ABB RobotStudio station: Solution1_20200531-184918.rsstn

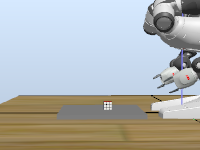
Station Solution1 (saved by RobotStudio 7.0.8746.631)
Controller IRB
  mechanical unit ROB_R: IRB14000_0.5_0.5_R, 6 joints, base frame (0, 0, 0) mm
  mechanical unit ROB_R_7: IRB14000_0.5_0.5_R, 1 joints, base frame (0, 0, 0) mm
  mechanical unit ROB_L: IRB14000_0.5_0.5_L, 6 joints, base frame (0, 0, 0) mm
  mechanical unit ROB_L_7: IRB14000_0.5_0.5_L, 1 joints, base frame (0, 0, 0) mm
Layout (positions relative to the parent item):
  - IRB14000_0.5_0.5 [mechanism, from Robots\IRB14000_0.5_0.5__01.rslib] at (0, 0, 0) mm
  - IRB14000_0.5_0.5_R [mechanism, from Robots\IRB14000_0.5_0.5__01.rslib] at (0, 0, 0) mm; joint values [0, -2.2689, -2.3562, 0.5236, 0, 0.6981, 0] (rad or m)
  - IRB14000_0.5_0.5_L [mechanism, from Robots\IRB14000_0.5_0.5__01.rslib] at (0, 0, 0) mm; joint values [0, -2.2689, 2.3562, 0.5236, 0, 0.6981, 0] (rad or m)
  - RightGripper [mechanism, from Tools\ABB_Smart_Gripper_Servo_Camera_Fingers.rslib] at (-9.58, -182.61, 198.63) mm, rotated rx 179.34 ry -63.63 rz 15.45 deg; joint values [0.025] (rad or m)
  - LeftGripper [mechanism, from Tools\ABB_Smart_Gripper_Servo_Camera_Fingers.rslib] at (-9.58, 182.61, 198.63) mm, rotated rx -179.34 ry -63.63 rz -15.45 deg; joint values [0.025] (rad or m)
  - floor [part]
  - table [part] at (0, -3.05, 0) mm
  - Cube [part] at (374.05, -18.3, 20.3) mm
Attachment: RightGripper is attached to IRB14000_0.5_0.5_R / Link7
Attachment: LeftGripper is attached to IRB14000_0.5_0.5_L / Link7
EventTableEntry 1735: Group=, Trigger=DO_CloseGripper 1736, Actions=[EventTableActionMechanicalPose 1737, EventTableActionAttach 1745], Comment=, ActivationMode=2, Cyclic=false
EventTableTriggerIO 1736: IOValue=[1], IRC5Controller=? -1, Operator=0, SignalSource=IRB 515
EventTableActionMechanicalPose 1737: VirtualSignal=SS_GripperIsClosed, Mechanism=RightGripper 1560, ToPoseName=PoseClose, VirtualSignalValue=[1]
EventTableEntry 1738: Group=, Trigger=DO_CloseGripper 1739, Actions=[EventTableActionMechanicalPose 1740, EventTableActionDetach 1747], Comment=, ActivationMode=2, Cyclic=false
EventTableTriggerIO 1739: IOValue=[0], IRC5Controller=? -1, Operator=0, SignalSource=IRB 515
EventTableActionMechanicalPose 1740: VirtualSignal=SS_GripperIsClosed, Mechanism=RightGripper 1560, ToPoseName=PoseOpen, VirtualSignalValue=[0]
EventTableEntry 1741: Group=, Trigger=NOP 1742, Actions=[DI_GripperIsClosed 1744], Comment=, ActivationMode=2, Cyclic=false
EventTableTriggerLogic 1742: layoutX=8, layoutY=16, Operand1=SS_GripperIsClosed 1743, Operand2=? -1, Operator=4, Delay=1000
EventTableTriggerIO 1743: IOValue=[-1], IRC5Controller=? -1, Operator=0, SignalSource=Solution1 1
EventTableActionIO 1744: IOValue=[-1], IRC5Controller=? -1, SignalTarget=IRB 515
EventTableActionAttach 1745: AttachmentParent=RightGripper 1560, AttachmentChild=Cube 1586, MountObject=false, Offset=[X=1, Y=0, Z=0, W=0, X=0, Y=1, Z=0, W=0, X=0, Y=0, Z=1, W=0, X=0, Y=0, Z=0, W=1], FlangeIndext=0, FindNearest=false
EventTableTriggerIO 1746: IOValue=[1], IRC5Controller=? -1, Operator=0, SignalSource=IRB 515
EventTableActionDetach 1747: AttachmentParent=RightGripper 1560, AttachmentChild=Cube 1586
EventTableTriggerIO 1748: IOValue=[0], IRC5Controller=? -1, Operator=0, SignalSource=IRB 515
EventTableTriggerLogic 1749: Operand1=SS_GripperIsClosed 1743, Operand2=? -1, Operator=4, Delay=1000
Station signals: DI SS_GripperIsClosed
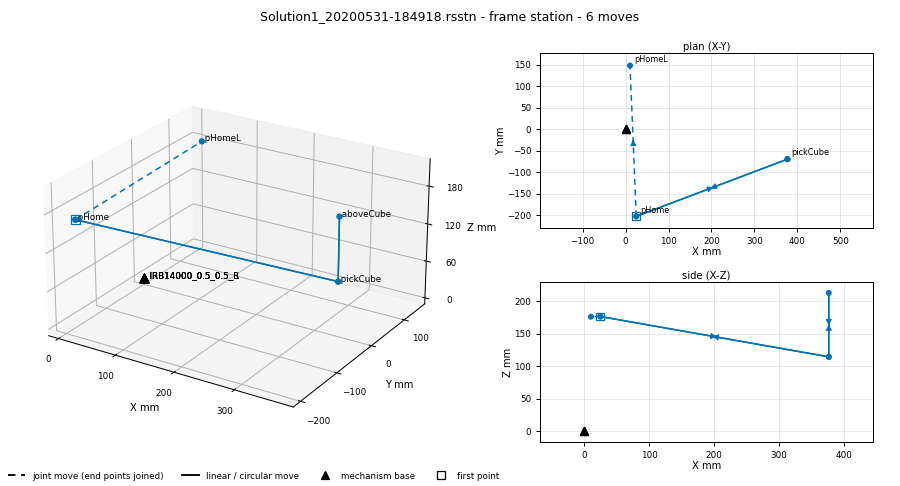
[picture p0: tool path of Solution1_20200531-184918.rsstn in frame station, 6 of 6 moves have a stored position in this frame; points joined in program order, loops and branches not executed]
Targets, tools, work objects and paths stored in the station, written as RAPID:
! task T_ROB_R
MODULE CalibData
  PERS tooldata Servo:=[TRUE,[[0,0,114.2],[1,0,0,0]],[0.229,[7.9,12.4,48.7],[1,0,0,0],0.00021,0.00023,0.00008]];
  PERS tooldata Camera:=[TRUE,[[-7.3,28.3,35.1],[0.5,-0.5,0.5,0.5]],[0.229,[7.9,12.4,48.7],[1,0,0,0],0.00021,0.00023,0.00008]];
  TASK PERS wobjdata Workobject_2:=[FALSE,TRUE,"",[[0,0,0],[1,0,0,0]],[[0,0,0],[1,0,0,0]]];
ENDMODULE

! task T_ROB_R
MODULE Module1
  CONST robtarget pHome:=[[24.971763923,-202.839465162,176.64502516],[0.07106331,0.248288947,-0.660142697,0.705346883],[0,0,0,4],[-101.964427132,9E+09,9E+09,9E+09,9E+09,9E+09]];
  CONST robtarget pickCube:=[[376.766775496,-69.805089288,114.555214565],[0.693258996,-0.185986842,-0.178114343,-0.673109307],[1,-1,0,4],[-118.392955921,9E+09,9E+09,9E+09,9E+09,9E+09]];
  CONST robtarget aboveCube:=[[376.76728936,-69.806028225,212.963720807],[0.717769789,0.002456743,0.004766394,-0.696259848],[1,-1,0,4],[-118.39295362,9E+09,9E+09,9E+09,9E+09,9E+09]];
  PROC main()
    MoveL pHome,v300,z100,Camera\WObj:=wobj0;
    MoveL pickCube,v300,fine,Camera\WObj:=Workobject_2;
    SetDO DO_CloseGripper,1;
    WaitDI DI_GripperIsClosed,1;
    MoveL aboveCube,v300,fine,Camera\WObj:=Workobject_2;
    MoveL pickCube,v300,fine,Camera\WObj:=Workobject_2;
    SetDO DO_CloseGripper,0;
    WaitDI DI_GripperIsClosed,0;
    MoveL pHome,v300,z100,Camera\WObj:=wobj0;
  ENDPROC
ENDMODULE

! task T_ROB_L
MODULE CalibData
  PERS tooldata Servo:=[TRUE,[[0,0,114.2],[1,0,0,0]],[0.229,[7.9,12.4,48.7],[1,0,0,0],0.00021,0.00023,0.00008]];
  PERS tooldata Camera:=[TRUE,[[-7.3,28.3,35.1],[0.5,-0.5,0.5,0.5]],[0.229,[7.9,12.4,48.7],[1,0,0,0],0.00021,0.00023,0.00008]];
  TASK PERS wobjdata Workobject_3:=[FALSE,TRUE,"",[[0,0,0],[1,0,0,0]],[[0,0,0],[1,0,0,0]]];
ENDMODULE

! task T_ROB_L
MODULE Module1
  CONST robtarget pHomeL:=[[10.457496534,148.132867885,176.35475559],[0.248288947,0.07106331,-0.705346883,0.660142697],[0,0,0,4],[101.964427132,9E+09,9E+09,9E+09,9E+09,9E+09]];
  PROC main()
    MoveJ pHomeL,v80,z100,Camera\WObj:=wobj0;
  ENDPROC
ENDMODULE

